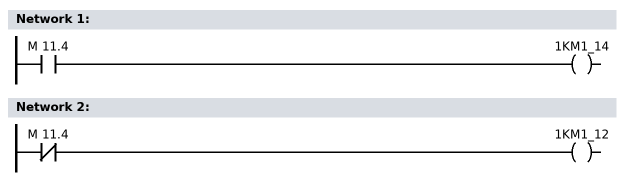
NETWORK
TITLE =
      A     "M 11.4";
      =     "1KM1_14";
NETWORK
TITLE =
      AN    "M 11.4";
      =     "1KM1_12";
END_FUNCTION

FUNCTION "FC 252" : VOID	// FC 252
VERSION : 0.1
BEGIN
// (block stored without names or comments; labels and parameter names are numbered)
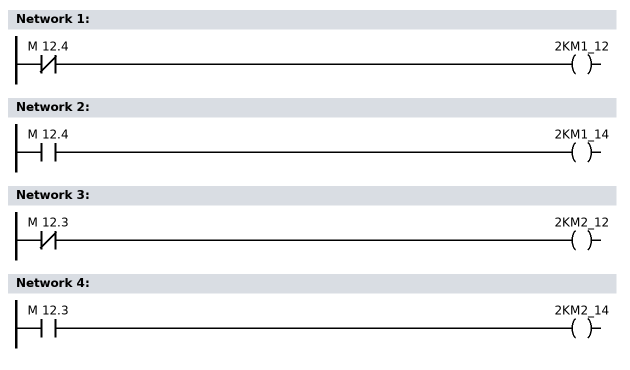
NETWORK
TITLE =
      AN    "M 12.4";
      =     "2KM1_12";
NETWORK
TITLE =
      A     "M 12.4";
      =     "2KM1_14";
NETWORK
TITLE =
      AN    "M 12.3";
      =     "2KM2_12";
NETWORK
TITLE =
      A     "M 12.3";
      =     "2KM2_14";
END_FUNCTION

FUNCTION "FC 253" : VOID	// FC 253
VERSION : 0.1
BEGIN
// (block stored without names or comments; labels and parameter names are numbered)
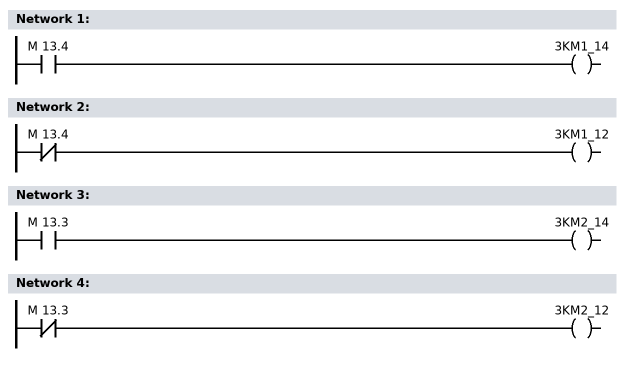
NETWORK
TITLE =
      A     "M 13.4";
      =     "3KM1_14";
NETWORK
TITLE =
      AN    "M 13.4";
      =     "3KM1_12";
NETWORK
TITLE =
      A     "M 13.3";
      =     "3KM2_14";
NETWORK
TITLE =
      AN    "M 13.3";
      =     "3KM2_12";
END_FUNCTION

FUNCTION "FC 254" : VOID	// FC 254
VERSION : 0.1
BEGIN
// (block stored without names or comments; labels and parameter names are numbered)
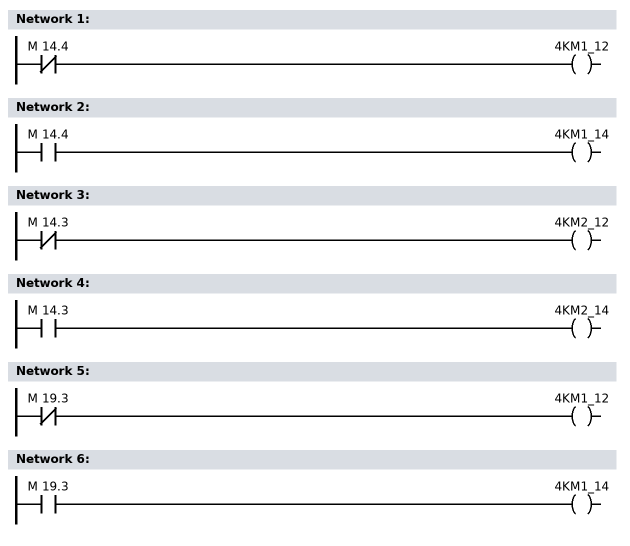
NETWORK
TITLE =
      AN    "M 14.4";
      =     "4KM1_12";
NETWORK
TITLE =
      A     "M 14.4";
      =     "4KM1_14";
NETWORK
TITLE =
      AN    "M 14.3";
      =     "4KM2_12";
NETWORK
TITLE =
      A     "M 14.3";
      =     "4KM2_14";
NETWORK
TITLE =
      AN    "M 19.3";
      =     "4KM1_12";
NETWORK
TITLE =
      A     "M 19.3";
      =     "4KM1_14";
END_FUNCTION

FUNCTION "FC 255" : VOID	// FC 255
VERSION : 0.1
BEGIN
// (block stored without names or comments; labels and parameter names are numbered)
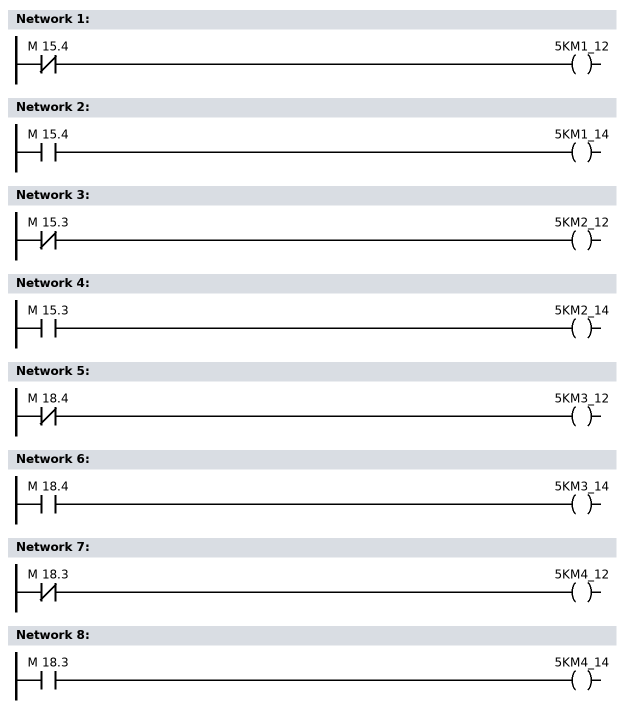
NETWORK
TITLE =
      AN    "M 15.4";
      =     "5KM1_12";
NETWORK
TITLE =
      A     "M 15.4";
      =     "5KM1_14";
NETWORK
TITLE =
      AN    "M 15.3";
      =     "5KM2_12";
NETWORK
TITLE =
      A     "M 15.3";
      =     "5KM2_14";
NETWORK
TITLE =
      AN    "M 18.4";
      =     "5KM3_12";
NETWORK
TITLE =
      A     "M 18.4";
      =     "5KM3_14";
NETWORK
TITLE =
      AN    "M 18.3";
      =     "5KM4_12";
NETWORK
TITLE =
      A     "M 18.3";
      =     "5KM4_14";
END_FUNCTION

FUNCTION "FC 256" : VOID	// FC 256
VERSION : 0.1
BEGIN
// (block stored without names or comments; labels and parameter names are numbered)
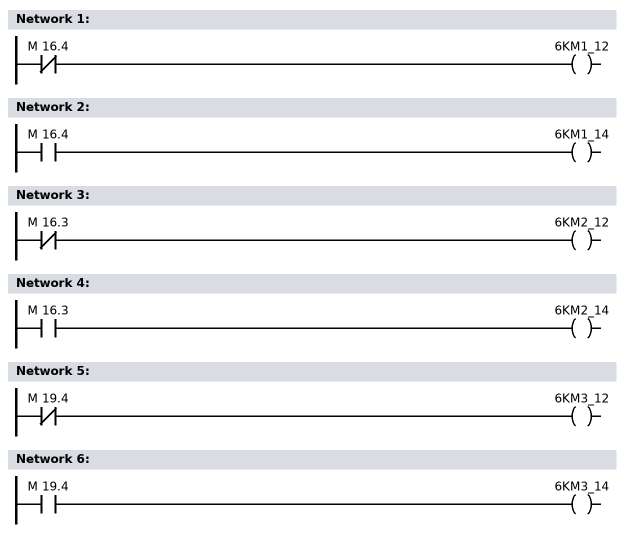
NETWORK
TITLE =
      AN    "M 16.4";
      =     "6KM1_12";
NETWORK
TITLE =
      A     "M 16.4";
      =     "6KM1_14";
NETWORK
TITLE =
      AN    "M 16.3";
      =     "6KM2_12";
NETWORK
TITLE =
      A     "M 16.3";
      =     "6KM2_14";
NETWORK
TITLE =
      AN    "M 19.4";
      =     "6KM3_12";
NETWORK
TITLE =
      A     "M 19.4";
      =     "6KM3_14";
END_FUNCTION

FUNCTION "FC 257" : VOID	// FC 257
VERSION : 0.1
BEGIN
// (block stored without names or comments; labels and parameter names are numbered)
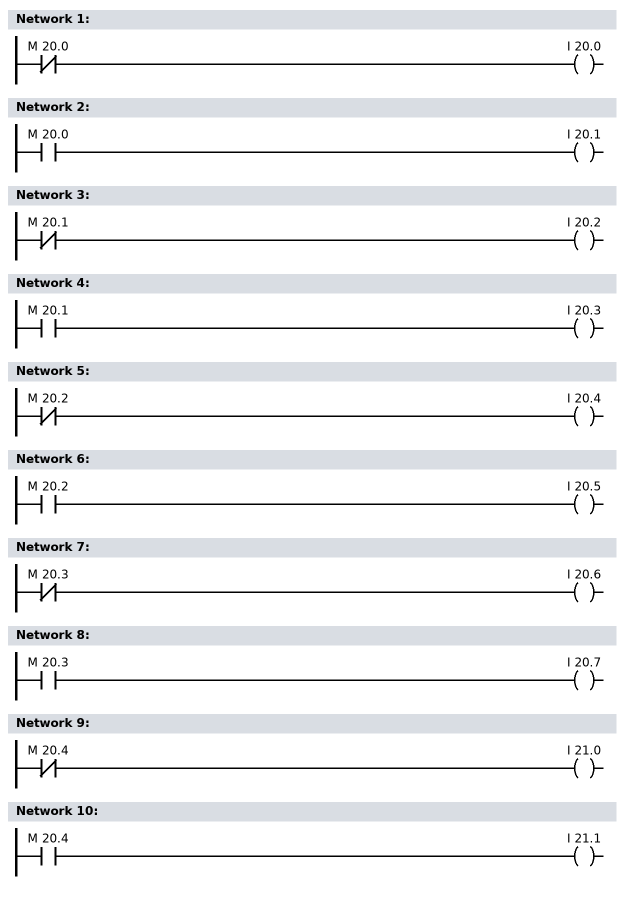
NETWORK
TITLE =
      AN    "M 20.0";
      =     I 20.0;
NETWORK
TITLE =
      A     "M 20.0";
      =     I 20.1;
NETWORK
TITLE =
      AN    "M 20.1";
      =     I 20.2;
NETWORK
TITLE =
      A     "M 20.1";
      =     I 20.3;
NETWORK
TITLE =
      AN    "M 20.2";
      =     I 20.4;
NETWORK
TITLE =
      A     "M 20.2";
      =     I 20.5;
NETWORK
TITLE =
      AN    "M 20.3";
      =     I 20.6;
NETWORK
TITLE =
      A     "M 20.3";
      =     I 20.7;
NETWORK
TITLE =
      AN    "M 20.4";
      =     I 21.0;
NETWORK
TITLE =
      A     "M 20.4";
      =     I 21.1;
END_FUNCTION

DATA_BLOCK "DB 126"	// DB 126
AUTHOR : ICom
FAMILY : DIAGNOSE
VERSION : 0.0
"PNIODiag"
BEGIN
END_DATA_BLOCK

DATA_BLOCK "DB 127"	// DB 127
AUTHOR : ICom
FAMILY : DIAGNOSE
VERSION : 0.0
"STATDiag"
BEGIN
END_DATA_BLOCK

DATA_BLOCK "DB 208"	// DB 208
AUTHOR : SIMATIC
FAMILY : EA_DIS
VERSION : 0.0
BEGIN
// 44 bytes; values not shown
END_DATA_BLOCK

DATA_BLOCK "DB 228"	// DB 228
AUTHOR : SIMATIC
FAMILY : EA_DIS
VERSION : 0.0
BEGIN
// 62 bytes; values not shown
END_DATA_BLOCK

ORGANIZATION_BLOCK "CYCL_EXC"	// OB 1
VERSION : 0.1
VAR_TEMP
  TEMP0 : BYTE ;
  TEMP1 : BYTE ;
  TEMP2 : BYTE ;
  TEMP3 : BYTE ;
  TEMP4 : BYTE ;
  TEMP5 : BYTE ;
  TEMP6 : INT ;
  TEMP7 : INT ;
  TEMP8 : INT ;
  TEMP9 : DATE_AND_TIME ;
END_VAR
BEGIN
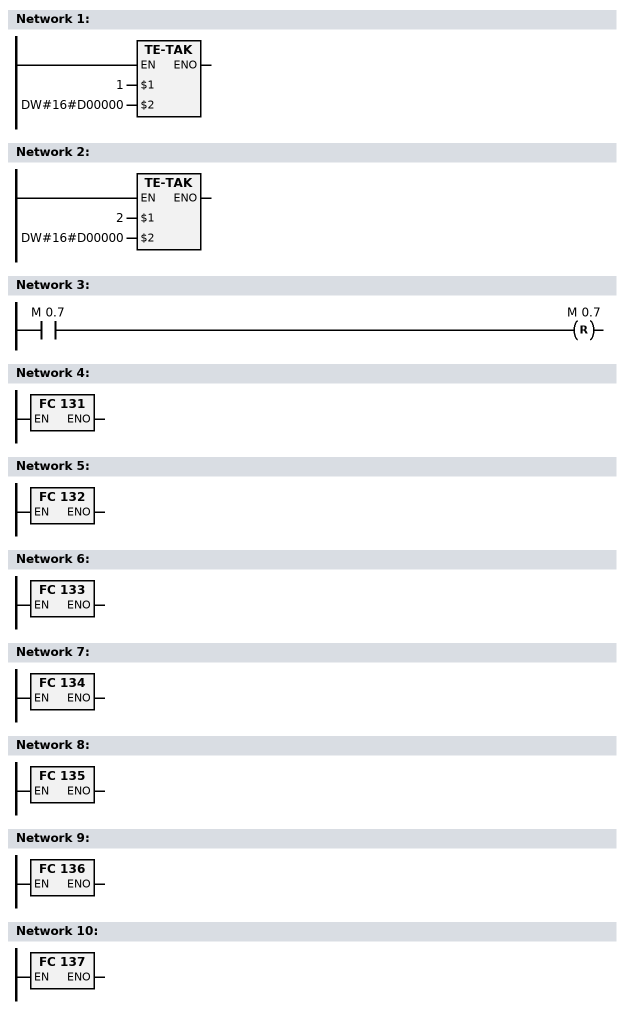
NETWORK
TITLE =
      CALL  "TE-TAK" (
           $1                       := 1,
           $2                       := DW#16#D00000);
      NOP   0;
NETWORK
TITLE =
      CALL  "TE-TAK" (
           $1                       := 2,
           $2                       := DW#16#D00000);
      NOP   0;
NETWORK
TITLE =
      A     "M 0.7";
      R     "M 0.7";
NETWORK
TITLE =
      CALL  "FC 131";
      NOP   0;
NETWORK
TITLE =
      CALL  "FC 132";
      NOP   0;
NETWORK
TITLE =
      CALL  "FC 133";
      NOP   0;
NETWORK
TITLE =
      CALL  "FC 134";
      NOP   0;
NETWORK
TITLE =
      CALL  "FC 135";
      NOP   0;
NETWORK
TITLE =
      CALL  "FC 136";
      NOP   0;
NETWORK
TITLE =
      CALL  "FC 137";
      NOP   0;
END_ORGANIZATION_BLOCK

ORGANIZATION_BLOCK "CYC_INT5"	// OB 35
VERSION : 0.1
BEGIN
// (block stored without names or comments; labels and parameter names are numbered)
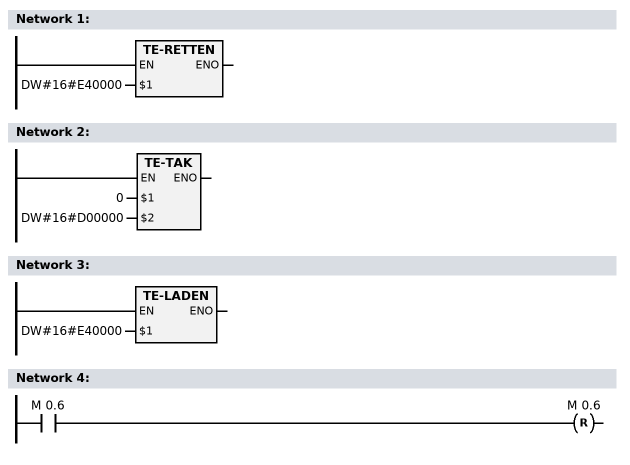
NETWORK
TITLE =
      CALL  "TE-RETTEN" (
           $1                       := DW#16#E40000);
      NOP   0;
NETWORK
TITLE =
      CALL  "TE-TAK" (
           $1                       := 0,
           $2                       := DW#16#D00000);
      NOP   0;
NETWORK
TITLE =
      CALL  "TE-LADEN" (
           $1                       := DW#16#E40000);
      NOP   0;
NETWORK
TITLE =
      A     "M 0.6";
      R     "M 0.6";
END_ORGANIZATION_BLOCK

ORGANIZATION_BLOCK "CYCL_FLT"	// OB 80
AUTHOR : SIMATIC
FAMILY : S7_300
NAME : TE_0B80
VERSION : 0.1
BEGIN
// (block stored without names or comments; labels and parameter names are numbered)
NETWORK
TITLE =
END_ORGANIZATION_BLOCK

ORGANIZATION_BLOCK "I/O_FLT1"	// OB 82
AUTHOR : SIMATIC
FAMILY : S7_300
NAME : TE_OB82
VERSION : 0.1
BEGIN
// (block stored without names or comments; labels and parameter names are numbered)
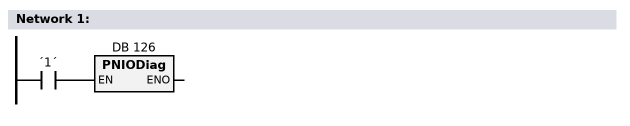
NETWORK
TITLE =
      A     "´1´";
      JNB   M001;
      CALL  "PNIODiag" , "DB 126";
M001: NOP   0;
END_ORGANIZATION_BLOCK

ORGANIZATION_BLOCK "OBNL_FLT"	// OB 85
AUTHOR : SIMATIC
FAMILY : S7_300
NAME : TE_OB85
VERSION : 0.1
BEGIN
// (block stored without names or comments; labels and parameter names are numbered)
END_ORGANIZATION_BLOCK

ORGANIZATION_BLOCK "RACK_FLT"	// OB 86
AUTHOR : SIMATIC
FAMILY : S7_300
NAME : TE_OB86
VERSION : 0.1
BEGIN
// (block stored without names or comments; labels and parameter names are numbered)
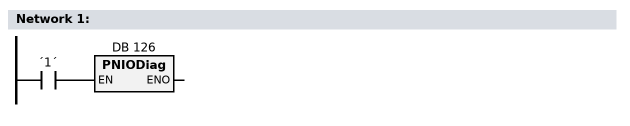
NETWORK
TITLE =
      A     "´1´";
      JNB   M001;
      CALL  "PNIODiag" , "DB 126";
M001: NOP   0;
END_ORGANIZATION_BLOCK

ORGANIZATION_BLOCK "COMM_FLT"	// OB 87
AUTHOR : SIMATIC
FAMILY : S7_300
NAME : TE_OB87
VERSION : 0.1
BEGIN
// (block stored without names or comments; labels and parameter names are numbered)
END_ORGANIZATION_BLOCK

ORGANIZATION_BLOCK "COMPLETE RESTART"	// OB 100
AUTHOR : SIMATIC
FAMILY : S7_300
NAME : TE_OB100
VERSION : 0.1
BEGIN
// (block stored without names or comments; labels and parameter names are numbered)
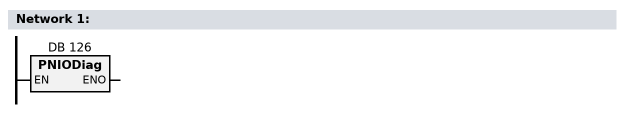
NETWORK
TITLE =
      CALL  "PNIODiag" , "DB 126";
      NOP   0;
END_ORGANIZATION_BLOCK

ORGANIZATION_BLOCK "PROG_ERR"	// OB 121
AUTHOR : SIMATIC
FAMILY : S7_300
NAME : TE_OB121
VERSION : 0.1
BEGIN
// (block stored without names or comments; labels and parameter names are numbered)
END_ORGANIZATION_BLOCK

ORGANIZATION_BLOCK "MOD_ERR"	// OB 122
AUTHOR : SIMATIC
FAMILY : S7_300
NAME : TE_OB122
VERSION : 0.1
BEGIN
// (block stored without names or comments; labels and parameter names are numbered)
END_ORGANIZATION_BLOCK
